{attribute 'GeneratedUsingTerminal: AT2050-0500-0019'}
{attribute addProperty BoxType "AT2050-0500-0019"}
{attribute addProperty Id "A_0094_AT2021_5250_0018_AT2021_5250AT2021_01D6DEDF80"}
{attribute addProperty CRC "2268875395"}
{attribute addProperty Size "80"}
TYPE A_0050_AT2050_0500_0019_873C4A83 EXTENDS AT2050_86175B41 :
STRUCT
	{attribute addProperty Name "A_0094_AT2021_5250_0018_AT2021_5250"}
	A_0094_AT2021_5250_0018_AT2021_5250 : AT2021_01D6DEDF;
END_STRUCT
END_TYPE

(* stored: Version 1.2.0.0, ProductVersion 3.1.4024.9
   DUT A_0050_AT2050_0500_0019_873C4A83: Id {cf1ae48e-7693-4dbc-91d4-cdef267d968e} *)
